Staubli VAL3: link_it.pgx

public program link_it(string x_sName)
begin
  // link the point
  link(tTraj[x_sName].pO,world)
  link(tTraj[x_sName].pX,world)
  link(tTraj[x_sName].pY,world)
  link(tTraj[x_sName].fFrame,world)
  link(tTraj[x_sName].pPointMove,tTraj[x_sName].fFrame)
  // put the base config
end
